FUNCTION_BLOCK E_LDU (* Event-driven Workpiece Load/Unload Model *)
  (* Standard: 61499-1; Function: GUI; Type: Selection; Description: Color selection *)
  (* Version 0.2, 2005-06-01, JHC, Holobloc Inc, Recompiled with new emitter. *)
  (* Version 0.1, 2004-10-18, JHC, Rockwell Automation, Derived from E_SEL_COLOR. *)
  (* Version 0.0, 2004-09-25, JHC, Rockwell Automation, Derived from E_SEL_COLOR. *)
  (* Compiler header: package fb.rt.mva; *)
  (* Compiler Java Sun JDK 1.4.2 *)
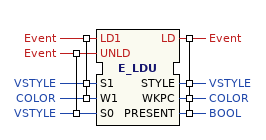
  EVENT_INPUT
    LD1 WITH S1, W1; (* Load Workpiece 1 *)
    UNLD WITH S0; (* Unload *)
  END_EVENT
  EVENT_OUTPUT
    LD WITH STYLE, WKPC, PRESENT; (* Load Command *)
  END_EVENT
  VAR_INPUT
    S1 : VSTYLE; (* Workpiece 1 Style *)
    W1 : COLOR; (* Workpiece 1 Color *)
    S0 : VSTYLE; (* Unloaded style *)
  END_VAR
  VAR_OUTPUT
    STYLE : VSTYLE; (* Workpiece Style *)
    WKPC : COLOR; (* Workpiece Color *)
    PRESENT : BOOL; (* Workpiece Present *)
  END_VAR
  ALGORITHM LD1 IN Java: (* Load Workpiece 1 *)
STYLE.value=S1.value;
WKPC.value=W1.value;
PRESENT.value = true;
LD.serviceEvent(this);
  END_ALGORITHM
  ALGORITHM UNLD IN Java: (* Unload Workpiece *)
STYLE.value = S0.value;
PRESENT.value = false;
LD.serviceEvent(this);
  END_ALGORITHM
END_FUNCTION_BLOCK
